(* IEC 61131-3 sources: CodesysTest/alpha/export/FBs/Unused/MotorizedSealFlattenersFB.pou, 3 files *)

(* ---- AutoMoveIn.m.st ---- *)
(*#-#-#-#-#-#-#-#-#-#---Declaration---#-#-#-#-#-#-#-#-#-#-#-#-#*)

METHOD AutoMoveIn : BOOL
VAR_INPUT
END_VAR
(*#-#-#-#-#-#-#-#-#-#---Implementation---#-#-#-#-#-#-#-#-#-#-#-#-#*)

_amMoveIn := TRUE;

(* ---- AutoMoveToBagHolding.m.st ---- *)
(*#-#-#-#-#-#-#-#-#-#---Declaration---#-#-#-#-#-#-#-#-#-#-#-#-#*)

METHOD AutoMoveToBagHolding
VAR_INPUT
END_VAR
(*#-#-#-#-#-#-#-#-#-#---Implementation---#-#-#-#-#-#-#-#-#-#-#-#-#*)

_amMoveInToBagHolding := TRUE;

(* ---- ClearCommands.m.st ---- *)
(*#-#-#-#-#-#-#-#-#-#---Declaration---#-#-#-#-#-#-#-#-#-#-#-#-#*)

METHOD PRIVATE ClearCommands
VAR_INPUT
END_VAR
(*#-#-#-#-#-#-#-#-#-#---Implementation---#-#-#-#-#-#-#-#-#-#-#-#-#*)

// Clear all commands from auto mode
_amMoveOut := FALSE;
_amMoveClearance := FALSE;
_amMoveInToBagHolding := FALSE;
_amMoveIn := FALSE;
